TEXTLIST TL_E_MOVER_SELECTOR
  0 = 'SELECT_MOVER_INDEX'
  1 = 'SELECT_MOVER_AXIS_ID'
   = ''
END_TEXTLIST

(* stored: Version 1.1.0.1
   TextList TL_E_MOVER_SELECTOR: Id {af08a30b-ad9a-4f52-a5b7-822d4558a047} *)
